TYPE MillimeterPerSecondSquared : LREAL;
END_TYPE

(* stored: Version 1.1.0.1, ProductVersion 3.1.4024.12
   DUT MillimeterPerSecondSquared: Id {2cb90d29-1cfd-4828-abab-08d141b5a473} *)
